(* CoDeSys 2.3 export: ST_PumpInterface.exp *)

(* Data type in Pump *)
(* ёЭвХадХЩб ЭРбЮбР *)
TYPE ST_PumpInterface :
STRUCT
    (* ІеЮФл *)
    stCommands : ST_PumpCommands;
    stProcessData : ST_PumpProcessData;
    stFCModbusIn : ST_FC_ModbusInterface;
    xExternalInterlock : BOOL;
    
    (* ІлеЮФл *)
    xReady : BOOL;
    xRunning : BOOL;
    xFault : BOOL;
    xWarning : BOOL;
    eState : E_PumpState;
    eMode : E_PumpMode;
    eFaultClass : E_PumpFaultClass;
    stDiagnostics : ST_PumpDiagnostics;
    stFCModbusOut : ST_FC_ModbusInterface;
END_STRUCT
END_TYPE
